// TwinCAT 3 PLC project StandardPLCProject
// ProgramVersion: 3.1.4024.0
// libraries:
//   Tc2_Standard, * (Beckhoff Automation GmbH)
//   Tc2_System, * (Beckhoff Automation GmbH)
//   Tc3_Module, * (Beckhoff Automation GmbH)
// project tree:
//   / PlcTask.TcTTO
//   POUs/ MAIN.TcPOU
// real-time tasks:
//   TASK PlcTask: cycle T#10ms, priority 6, ADS port 350
// I/O:
//   DEVICE Device 2 (EtherCAT), AmsNetId 172.24.112.1.3.1
//     Term 1 (EK1100) [EK1100 EtherCAT Coupler (2A E-Bus)]
//       Term 2 (EL1008) [EL1008 8Ch. Dig. Input 24V, 3ms]
//       Term 3 (EL2008) [EL2008 8Ch. Dig. Output 24V, 0.5A]
//       Term 4 (EL3002) [EL3002 2Ch. Ana. Input +/-10V]
//       Term 5 (EL3202) [EL3202 2Ch. Ana. Input PT100 (RTD)]
//       Term 6 (EL9011) [EL9011 End Terminal]
// variable links:
//   StandardPLCProject/StandardPLCProject Instance <-> Device 2 (EtherCAT)/Term 1 (EK1100)/Term 3 (EL2008)
//     PlcTask Outputs/MAIN.bLampa <-> Channel 1/Output

CONFIGURATION StandardPLCProject
    RESOURCE PLC ON TwinCAT3
        TASK PlcTask(INTERVAL := T#10ms, PRIORITY := 20);
        PROGRAM MAIN WITH PlcTask : MAIN;
    END_RESOURCE
END_CONFIGURATION

// ---- POUs/MAIN.TcPOU
PROGRAM MAIN
VAR
    fbTimer   : TON;         // Deklaracja naszego timera
    bMrugnij  : BOOL;        // Zmienna, która będzie migać (Prawda/Fałsz)
    tCzas     : TIME := T#1S; // Czas, co ile ma migać (1 sekunda)
END_VAR

// Wywołanie timera
// IN: wejście (jeśli TRUE, zaczyna liczyć)
// PT: Preset Time (zadany czas)
fbTimer(IN := NOT fbTimer.Q, PT := tCzas);

// Jeśli timer doliczył do końca (wyjście Q zrobiło się TRUE)
IF fbTimer.Q THEN
    bMrugnij := NOT bMrugnij; // Zmień stan zmiennej na przeciwny
END_IF

END_PROGRAM
